FUNCTION_BLOCK Single_LED_Controller (* Composite Function Block Type *)
  (* Standard: 61499-2 *)
  (* Version 0.0, 9/22/2026, macie, Schneider Electric, template *)
  PACKAGE Main;
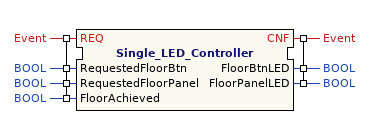
  EVENT_INPUT
    REQ WITH RequestedFloorBtn, FloorAchieved, RequestedFloorPanel; (* Normal Execution Request *)
  END_EVENT
  EVENT_OUTPUT
    CNF WITH FloorBtnLED, FloorPanelLED; (* Execution Confirmation *)
  END_EVENT
  VAR_INPUT
    RequestedFloorBtn : BOOL; (* Input event qualifier *)
    RequestedFloorPanel : BOOL;
    FloorAchieved : BOOL;
  END_VAR
  VAR_OUTPUT
    FloorBtnLED : BOOL; (* Output event qualifier *)
    FloorPanelLED : BOOL;
  END_VAR
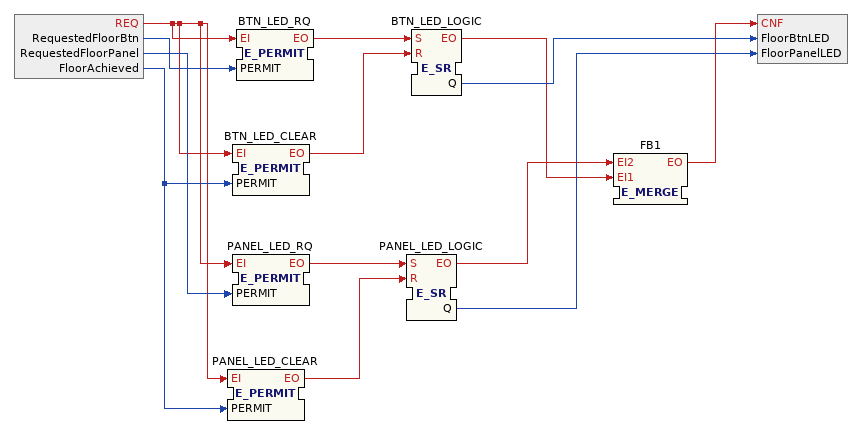
  FBS
    BTN_LED_LOGIC : E_SR;
    BTN_LED_RQ : E_PERMIT;
    BTN_LED_CLEAR : E_PERMIT;
    PANEL_LED_LOGIC : E_SR;
    PANEL_LED_RQ : E_PERMIT;
    PANEL_LED_CLEAR : E_PERMIT;
    FB1 : E_MERGE;
  END_FBS
  EVENT_CONNECTIONS
    BTN_LED_RQ.EO TO BTN_LED_LOGIC.S;
    BTN_LED_CLEAR.EO TO BTN_LED_LOGIC.R;
    REQ TO BTN_LED_RQ.EI;
    REQ TO BTN_LED_CLEAR.EI;
    PANEL_LED_RQ.EO TO PANEL_LED_LOGIC.S;
    PANEL_LED_CLEAR.EO TO PANEL_LED_LOGIC.R;
    REQ TO PANEL_LED_RQ.EI;
    REQ TO PANEL_LED_CLEAR.EI;
    PANEL_LED_LOGIC.EO TO FB1.EI2;
    FB1.EO TO CNF;
    BTN_LED_LOGIC.EO TO FB1.EI1;
  END_CONNECTIONS
  DATA_CONNECTIONS
    BTN_LED_LOGIC.Q TO FloorBtnLED;
    RequestedFloorBtn TO BTN_LED_RQ.PERMIT;
    FloorAchieved TO BTN_LED_CLEAR.PERMIT;
    RequestedFloorPanel TO PANEL_LED_RQ.PERMIT;
    PANEL_LED_LOGIC.Q TO FloorPanelLED;
    FloorAchieved TO PANEL_LED_CLEAR.PERMIT;
  END_CONNECTIONS
END_FUNCTION_BLOCK
